_CFC_ (* Continuous Function Chart, elements in execution order *)
#0 OR(SCHU_P2_3_UE2_T_RESET, SCHU_P2_3_SB)
#1 SEL(UE2_T_FILTER_ON, T#0ms, T#2s)
#2 fb_UE2_T:ISTOK_ANALOGVH(enable: TRUE, rawValue: SCHU_P2_3_UE2_AI1, reset: #0, enableLimitCtrl: enbleLimit, ctrlVoltage: NOT UE2_T_CVOLT, changeValueWithoutPower: TRUE, highRange: UE_T_HIGHRANGE, lowRange: UE_T_LOWRANGE, highLimit: SCHU_P2_3_UE_T_HIGHLIMIT, lowLimit: SCHU_P2_3_UE_T_LOWLIMIT, filterTime: #1, offset: ofset, delayEnable: TE_DELAY)
#3 SCHU_P2_3_UE2_T_VN <= #2.presentValue
#4 SCHU_P2_3_UE2_T_DOST <= #2.reliability
#5 SUB(SCHU_P2_3_UE2_T_UST, 0.6)
#6 fb_UE2_m_UST:ISTOK_LT(dost: #2.reliability, x: #2.presentValue, ust: #5, shkal: -, gist: 0.5)
#7 SCHU_P2_3_UE2_TE_M_UST <= #6.Xm
#8 SCHU_P2_3_UE2_TE_NM_UST <= #6.XmN
#9 ADD(SCHU_P2_3_UE2_T_UST, 0.6)
#10 fb_UE2_b_UST:ISTOK_GT(dost: #2.reliability, x: #2.presentValue, ust: #9, shkal: -, gist: 0.5)
#11 SCHU_P2_3_UE2_TE_B_UST <= #10.Xb
#12 SCHU_P2_3_UE2_TE_NB_UST <= #10.XbN
_END_CFC_
(* the same logic as Structured Text *)
fb_UE2_T(enable := TRUE, rawValue := SCHU_P2_3_UE2_AI1, reset := SCHU_P2_3_UE2_T_RESET OR SCHU_P2_3_SB, enableLimitCtrl := enbleLimit, ctrlVoltage := NOT UE2_T_CVOLT, changeValueWithoutPower := TRUE, highRange := UE_T_HIGHRANGE, lowRange := UE_T_LOWRANGE, highLimit := SCHU_P2_3_UE_T_HIGHLIMIT, lowLimit := SCHU_P2_3_UE_T_LOWLIMIT, filterTime := SEL(UE2_T_FILTER_ON, T#0ms, T#2s), offset := ofset, delayEnable := TE_DELAY);
SCHU_P2_3_UE2_T_VN := fb_UE2_T.presentValue;
SCHU_P2_3_UE2_T_DOST := fb_UE2_T.reliability;
fb_UE2_m_UST(dost := fb_UE2_T.reliability, x := fb_UE2_T.presentValue, ust := SCHU_P2_3_UE2_T_UST - 0.6, gist := 0.5);
SCHU_P2_3_UE2_TE_M_UST := fb_UE2_m_UST.Xm;
SCHU_P2_3_UE2_TE_NM_UST := fb_UE2_m_UST.XmN;
fb_UE2_b_UST(dost := fb_UE2_T.reliability, x := fb_UE2_T.presentValue, ust := SCHU_P2_3_UE2_T_UST + 0.6, gist := 0.5);
SCHU_P2_3_UE2_TE_B_UST := fb_UE2_b_UST.Xb;
SCHU_P2_3_UE2_TE_NB_UST := fb_UE2_b_UST.XbN;
END_PROGRAM

(* POU Input/AI/UE2_VL, CFC *)
PROGRAM UE2_VL
VAR
	fb_UE2_VL: ISTOK_ANALOGVH;
	ofset: REAL;
	fb_UE2_VLbUST: ISTOK_GT;
END_VAR
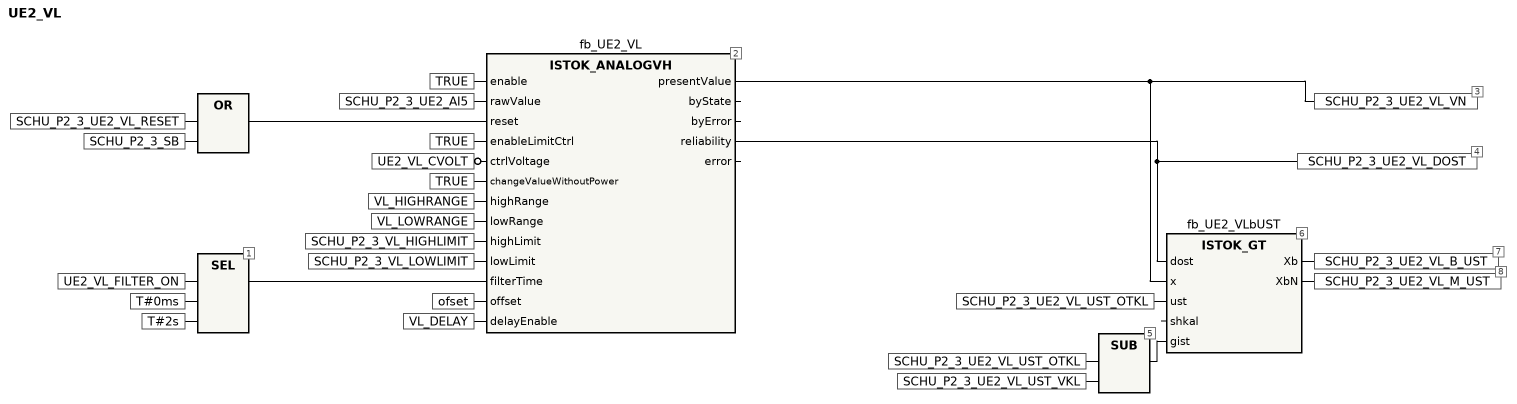
_CFC_ (* Continuous Function Chart, elements in execution order *)
#0 OR(SCHU_P2_3_UE2_VL_RESET, SCHU_P2_3_SB)
#1 SEL(UE2_VL_FILTER_ON, T#0ms, T#2s)
#2 fb_UE2_VL:ISTOK_ANALOGVH(enable: TRUE, rawValue: SCHU_P2_3_UE2_AI5, reset: #0, enableLimitCtrl: TRUE, ctrlVoltage: NOT UE2_VL_CVOLT, changeValueWithoutPower: TRUE, highRange: VL_HIGHRANGE, lowRange: VL_LOWRANGE, highLimit: SCHU_P2_3_VL_HIGHLIMIT, lowLimit: SCHU_P2_3_VL_LOWLIMIT, filterTime: #1, offset: ofset, delayEnable: VL_DELAY)
#3 SCHU_P2_3_UE2_VL_VN <= #2.presentValue
#4 SCHU_P2_3_UE2_VL_DOST <= #2.reliability
#5 SUB(SCHU_P2_3_UE2_VL_UST_OTKL, SCHU_P2_3_UE2_VL_UST_VKL)
#6 fb_UE2_VLbUST:ISTOK_GT(dost: #2.reliability, x: #2.presentValue, ust: SCHU_P2_3_UE2_VL_UST_OTKL, shkal: -, gist: #5)
#7 SCHU_P2_3_UE2_VL_B_UST <= #6.Xb
#8 SCHU_P2_3_UE2_VL_M_UST <= #6.XbN
_END_CFC_
(* the same logic as Structured Text *)
fb_UE2_VL(enable := TRUE, rawValue := SCHU_P2_3_UE2_AI5, reset := SCHU_P2_3_UE2_VL_RESET OR SCHU_P2_3_SB, enableLimitCtrl := TRUE, ctrlVoltage := NOT UE2_VL_CVOLT, changeValueWithoutPower := TRUE, highRange := VL_HIGHRANGE, lowRange := VL_LOWRANGE, highLimit := SCHU_P2_3_VL_HIGHLIMIT, lowLimit := SCHU_P2_3_VL_LOWLIMIT, filterTime := SEL(UE2_VL_FILTER_ON, T#0ms, T#2s), offset := ofset, delayEnable := VL_DELAY);
SCHU_P2_3_UE2_VL_VN := fb_UE2_VL.presentValue;
SCHU_P2_3_UE2_VL_DOST := fb_UE2_VL.reliability;
fb_UE2_VLbUST(dost := fb_UE2_VL.reliability, x := fb_UE2_VL.presentValue, ust := SCHU_P2_3_UE2_VL_UST_OTKL, gist := SCHU_P2_3_UE2_VL_UST_OTKL - SCHU_P2_3_UE2_VL_UST_VKL);
SCHU_P2_3_UE2_VL_B_UST := fb_UE2_VLbUST.Xb;
SCHU_P2_3_UE2_VL_M_UST := fb_UE2_VLbUST.XbN;
END_PROGRAM

(* POU Input/AI/UE3_T, CFC *)
PROGRAM UE3_T
VAR
	fb_UE3_T: ISTOK_ANALOGVH;
	ofset: REAL;
	fb_SCHU_P2_3_UE3_T_NEQ_UST: ISTOK_EQ;
	fb_UE3_m_UST: ISTOK_LT;
END_VAR
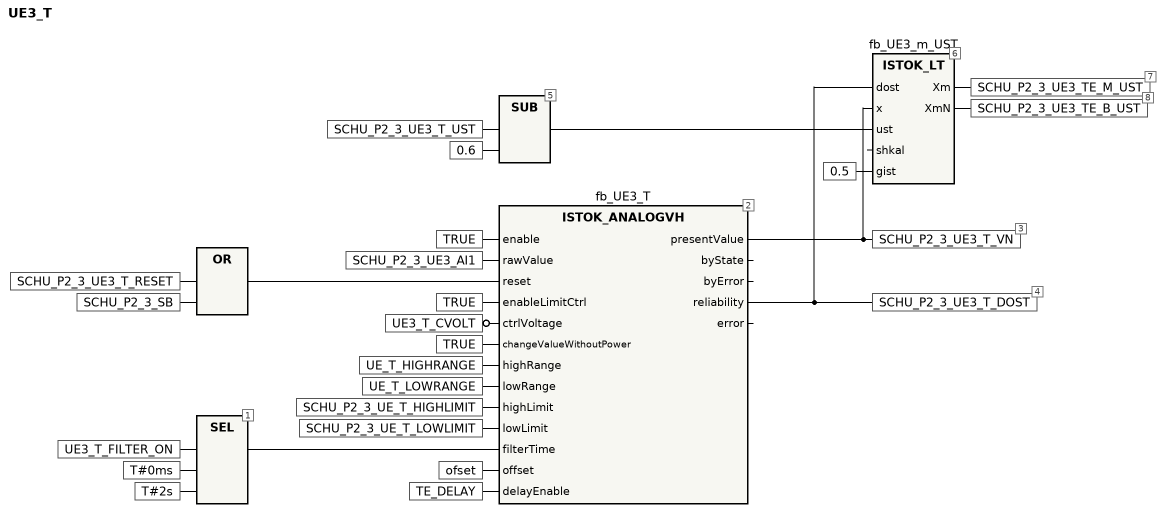
_CFC_ (* Continuous Function Chart, elements in execution order *)
#0 OR(SCHU_P2_3_UE3_T_RESET, SCHU_P2_3_SB)
#1 SEL(UE3_T_FILTER_ON, T#0ms, T#2s)
#2 fb_UE3_T:ISTOK_ANALOGVH(enable: TRUE, rawValue: SCHU_P2_3_UE3_AI1, reset: #0, enableLimitCtrl: TRUE, ctrlVoltage: NOT UE3_T_CVOLT, changeValueWithoutPower: TRUE, highRange: UE_T_HIGHRANGE, lowRange: UE_T_LOWRANGE, highLimit: SCHU_P2_3_UE_T_HIGHLIMIT, lowLimit: SCHU_P2_3_UE_T_LOWLIMIT, filterTime: #1, offset: ofset, delayEnable: TE_DELAY)
#3 SCHU_P2_3_UE3_T_VN <= #2.presentValue
#4 SCHU_P2_3_UE3_T_DOST <= #2.reliability
#5 SUB(SCHU_P2_3_UE3_T_UST, 0.6)
#6 fb_UE3_m_UST:ISTOK_LT(dost: #2.reliability, x: #2.presentValue, ust: #5, shkal: -, gist: 0.5)
#7 SCHU_P2_3_UE3_TE_M_UST <= #6.Xm
#8 SCHU_P2_3_UE3_TE_B_UST <= #6.XmN
_END_CFC_
(* the same logic as Structured Text *)
fb_UE3_T(enable := TRUE, rawValue := SCHU_P2_3_UE3_AI1, reset := SCHU_P2_3_UE3_T_RESET OR SCHU_P2_3_SB, enableLimitCtrl := TRUE, ctrlVoltage := NOT UE3_T_CVOLT, changeValueWithoutPower := TRUE, highRange := UE_T_HIGHRANGE, lowRange := UE_T_LOWRANGE, highLimit := SCHU_P2_3_UE_T_HIGHLIMIT, lowLimit := SCHU_P2_3_UE_T_LOWLIMIT, filterTime := SEL(UE3_T_FILTER_ON, T#0ms, T#2s), offset := ofset, delayEnable := TE_DELAY);
SCHU_P2_3_UE3_T_VN := fb_UE3_T.presentValue;
SCHU_P2_3_UE3_T_DOST := fb_UE3_T.reliability;
fb_UE3_m_UST(dost := fb_UE3_T.reliability, x := fb_UE3_T.presentValue, ust := SCHU_P2_3_UE3_T_UST - 0.6, gist := 0.5);
SCHU_P2_3_UE3_TE_M_UST := fb_UE3_m_UST.Xm;
SCHU_P2_3_UE3_TE_B_UST := fb_UE3_m_UST.XmN;
END_PROGRAM

(* POU Input/AI/UE3_VL, CFC *)
PROGRAM UE3_VL
VAR
	fb_UE3_VL: ISTOK_ANALOGVH;
	ofset: REAL;
	fb_SCHU_P2_3_UE3_VL_B_UST: ISTOK_GT;
END_VAR
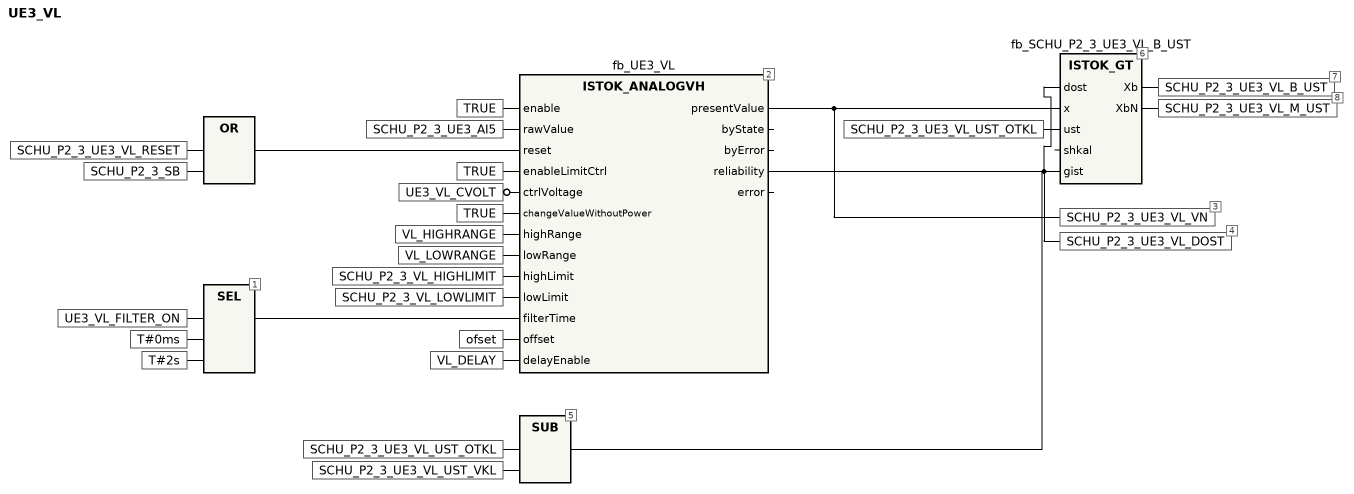
